// TIA Portal project "CMConstruccionesAutomatizacionHormigonera" (V16)

(* hardware
DEVICE "S7-1200 station_1"  S7-1200 Station
   slot 0: "Rack_0"  S7-1200 Rack  Rack  V1.0
   slot 1: "PLC_1"  CPU 1212C AC/DC/Rly  6ES7 212-1BE40-0XB0  V4.4
   slot 2: "DQ 8xRelay_1"  SM 1222 DQ8 x relay  6ES7 222-1HF32-0XB0  V2.0
*)

// ===== PLC "PLC_1"  CPU 1212C AC/DC/Rly =====

VAR_GLOBAL   // PLC tag table "Tabla de variables estándar"
   "Automatico" AT %I0.0 : Bool;
   "Sin Fin 1" AT %Q8.4 : Bool;
   "Start Cemento" AT %M0.0 : Bool;
   "Silo 1" AT %M0.1 : Bool;
   "Compuerta 1" AT %Q8.5 : Bool;
   "Silo 2" AT %M0.2 : Bool;
   "Compuerta 2" AT %Q0.5 : Bool;
   "Cemento listo" AT %M0.3 : Bool;
   "Input_Encoder" AT %ID1000 : DInt;
   "Comp Cemento listo" AT %Q8.0 : Bool;
   "Condiciones Cemento" AT %M0.4 : Bool;
   "Start Descarga" AT %M0.5 : Bool;
   "Piedra Listo" AT %M0.6 : Bool;
   "Compuerta 3" AT %Q0.0 : Bool;
   "Tag_1" AT %M0.7 : Bool;
   "Condiciones Piedra" AT %M3.0 : Bool;
   "Condiciones Arena" AT %M2.1 : Bool;
   "Compuerta 4" AT %Q0.2 : Bool;
   "Arena listo" AT %M2.2 : Bool;
   "Direccion encoder" AT %I0.2 : Bool;
   "Paso Piedra" AT %M2.3 : Bool;
   "Paso Arena" AT %M1.4 : Bool;
   "Start Agua" AT %M2.5 : Bool;
   "Condiciones Agua" AT %M1.6 : Bool;
   "Agua listo" AT %M1.7 : Bool;
   "Compresor" AT %Q8.3 : Bool;
   "Banda" AT %Q8.1 : Bool;
   "Agua" AT %Q8.2 : Bool;
   "Compuerta 5" AT %Q0.3 : Bool;
   "Paso Agua" AT %M2.0 : Bool;
   "System_Byte" AT %MB1 : Byte;
   "FirstScan" AT %M1.0 : Bool;
   "DiagStatusUpdate" AT %M1.1 : Bool;
   "AlwaysTRUE" AT %M1.2 : Bool;
   "AlwaysFALSE" AT %M1.3 : Bool;
   "System_Byte(1)" AT %MB2 : Byte;
   "Pulsos" AT %MD4 : DInt;
   "STATUS" AT %MW8 : Word;
   "Contador Agua" AT %I0.3 : Bool;
   "Salida Contador Agua" AT %MW10 : Word;
   "Ingreso Contador Agua" AT %MW12 : Word;
   "Compuerta 6" AT %Q0.4 : Bool;
   "reiniciar cemento" AT %M3.1 : Bool;
   "Tag_2" AT %M3.2 : Bool;
   "reiniciar aridos" AT %M3.3 : Bool;
   "Tag_3" AT %M3.4 : Bool;
   "arena paso" AT %M3.5 : Bool;
   "TiempoArena" AT %M3.6 : Bool;
   "fin cemento" AT %M3.7 : Bool;
   "tiempo banda" AT %M14.0 : Bool;
   "reserva" AT %M14.1 : Bool;
   "Compresor listo" AT %M14.2 : Bool;
   "fin aridos" AT %M14.3 : Bool;
   "Agua completa" AT %M14.4 : Bool;
   "Piedra 2" AT %Q0.1 : Bool;
END_VAR

// folder: System blocks/Program resources

DATA_BLOCK "IEC_Timer_0_DB"   // DB1
{ S7_Optimized_Access := 'TRUE' }
AUTHOR : Simatic
FAMILY : IEC
NAME : IEC_TMR
VERSION : 1.0
// stored: InstanceOfName IEC_TIMER
"IEC_TIMER"
BEGIN
END_DATA_BLOCK

DATA_BLOCK "IEC_Timer_0_DB_1"   // DB2
{ S7_Optimized_Access := 'TRUE' }
AUTHOR : Simatic
FAMILY : IEC
NAME : IEC_TMR
VERSION : 1.0
// stored: InstanceOfName IEC_TIMER
"IEC_TIMER"
BEGIN
END_DATA_BLOCK

DATA_BLOCK "IEC_Timer_0_DB_2"   // DB3
{ S7_Optimized_Access := 'TRUE' }
AUTHOR : Simatic
FAMILY : IEC
NAME : IEC_TMR
VERSION : 1.0
// stored: InstanceOfName IEC_TIMER
"IEC_TIMER"
BEGIN
END_DATA_BLOCK

DATA_BLOCK "IEC_Timer_0_DB_3"   // DB4
{ S7_Optimized_Access := 'TRUE' }
AUTHOR : Simatic
FAMILY : IEC
NAME : IEC_TMR
VERSION : 1.0
// stored: InstanceOfName IEC_TIMER
"IEC_TIMER"
BEGIN
END_DATA_BLOCK

DATA_BLOCK "IEC_Counter_0_DB"   // DB5
{ S7_Optimized_Access := 'TRUE' }
AUTHOR : Simatic
FAMILY : IEC
NAME : CNTR
VERSION : 1.0
// stored: InstanceOfName IEC_COUNTER
"IEC_COUNTER"
BEGIN
END_DATA_BLOCK

DATA_BLOCK "IEC_Timer_0_DB_4"   // DB6
{ S7_Optimized_Access := 'TRUE' }
AUTHOR : Simatic
FAMILY : IEC
NAME : IEC_TMR
VERSION : 1.0
// stored: InstanceOfName IEC_TIMER
"IEC_TIMER"
BEGIN
END_DATA_BLOCK

DATA_BLOCK "IEC_Timer_0_DB_5"   // DB7
{ S7_Optimized_Access := 'TRUE' }
AUTHOR : Simatic
FAMILY : IEC
NAME : IEC_TMR
VERSION : 1.0
// stored: InstanceOfName IEC_TIMER
"IEC_TIMER"
BEGIN
END_DATA_BLOCK

DATA_BLOCK "IEC_Timer_0_DB_6"   // DB8
{ S7_Optimized_Access := 'TRUE' }
AUTHOR : Simatic
FAMILY : IEC
NAME : IEC_TMR
VERSION : 1.0
// stored: InstanceOfName IEC_TIMER
"IEC_TIMER"
BEGIN
END_DATA_BLOCK

DATA_BLOCK "IEC_Timer_0_DB_7"   // DB9
{ S7_Optimized_Access := 'TRUE' }
AUTHOR : Simatic
FAMILY : IEC
NAME : IEC_TMR
VERSION : 1.0
// stored: InstanceOfName IEC_TIMER
"IEC_TIMER"
BEGIN
END_DATA_BLOCK

DATA_BLOCK "IEC_Timer_0_DB_8"   // DB10
{ S7_Optimized_Access := 'TRUE' }
AUTHOR : Simatic
FAMILY : IEC
NAME : IEC_TMR
VERSION : 1.0
// stored: InstanceOfName IEC_TIMER
"IEC_TIMER"
BEGIN
END_DATA_BLOCK

// folder: (top level)

ORGANIZATION_BLOCK "Main"   // OB1, LAD, ProgramCycle
TITLE = "Main Program Sweep (Cycle)"
{ S7_Optimized_Access := 'TRUE' }
VERSION : 0.1
   VAR_INPUT
      Initial_Call : Bool;   // Initial call of this OB
      Remanence : Bool;   // =True, if remanent data are available
   END_VAR
   VAR_TEMP   // added for the SCL form of the ladder/FBD networks
      _w1 : Bool;
      _w2 : Bool;
   END_VAR
BEGIN

REGION Network 1
   // Proceso Cemento
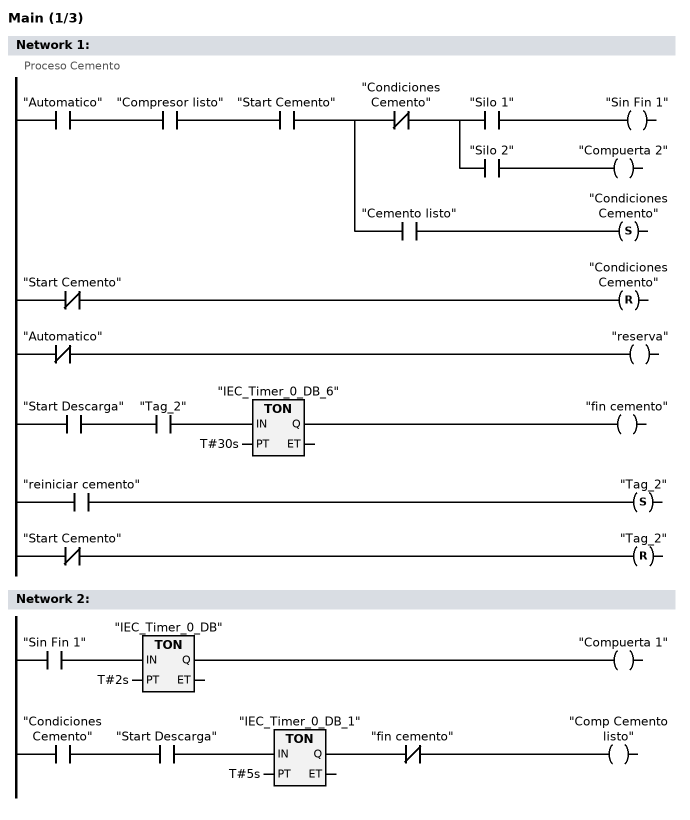
   #_w1 := "Automatico" AND "Compresor listo" AND "Start Cemento";
   #_w2 := #_w1 AND NOT "Condiciones Cemento";
   "Sin Fin 1" := #_w2 AND "Silo 1";
   "Compuerta 2" := #_w2 AND "Silo 2";
   IF #_w1 AND "Cemento listo" THEN "Condiciones Cemento" := TRUE; END_IF;
   IF NOT "Start Cemento" THEN "Condiciones Cemento" := FALSE; END_IF;
   "reserva" := NOT "Automatico";
   "IEC_Timer_0_DB_6".TON(IN := "Start Descarga" AND "Tag_2", PT := T#30s);
   "fin cemento" := "IEC_Timer_0_DB_6".Q;
   IF "reiniciar cemento" THEN "Tag_2" := TRUE; END_IF;
   IF NOT "Start Cemento" THEN "Tag_2" := FALSE; END_IF;
END_REGION

REGION Network 2
   "IEC_Timer_0_DB".TON(IN := "Sin Fin 1", PT := T#2s);
   "Compuerta 1" := "IEC_Timer_0_DB".Q;
   "IEC_Timer_0_DB_1".TON(IN := "Condiciones Cemento" AND "Start Descarga", PT := T#5s);
   "Comp Cemento listo" := "IEC_Timer_0_DB_1".Q AND NOT "fin cemento";
END_REGION

REGION Network 3
   // Proceso Aridos
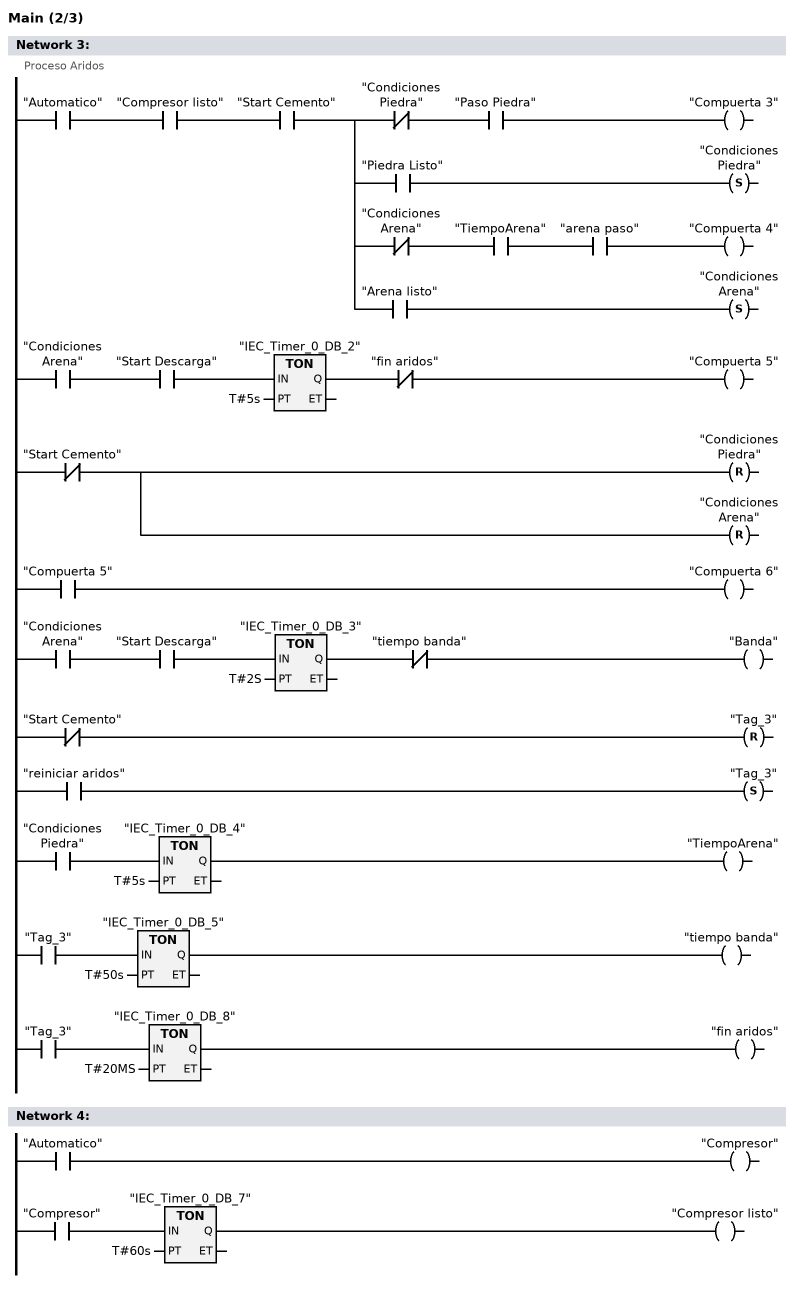
   #_w1 := "Automatico" AND "Compresor listo" AND "Start Cemento";
   "Compuerta 3" := #_w1 AND NOT "Condiciones Piedra" AND "Paso Piedra";
   IF #_w1 AND "Piedra Listo" THEN "Condiciones Piedra" := TRUE; END_IF;
   "Compuerta 4" := #_w1 AND NOT "Condiciones Arena" AND "TiempoArena" AND "arena paso";
   IF #_w1 AND "Arena listo" THEN "Condiciones Arena" := TRUE; END_IF;
   "IEC_Timer_0_DB_2".TON(IN := "Condiciones Arena" AND "Start Descarga", PT := T#5s);
   "Compuerta 5" := "IEC_Timer_0_DB_2".Q AND NOT "fin aridos";
   IF NOT "Start Cemento" THEN
       "Condiciones Piedra" := FALSE;
       "Condiciones Arena" := FALSE;
   END_IF;
   "Compuerta 6" := "Compuerta 5";
   "IEC_Timer_0_DB_3".TON(IN := "Condiciones Arena" AND "Start Descarga", PT := T#2S);
   "Banda" := "IEC_Timer_0_DB_3".Q AND NOT "tiempo banda";
   IF NOT "Start Cemento" THEN "Tag_3" := FALSE; END_IF;
   IF "reiniciar aridos" THEN "Tag_3" := TRUE; END_IF;
   "IEC_Timer_0_DB_4".TON(IN := "Condiciones Piedra", PT := T#5s);
   "TiempoArena" := "IEC_Timer_0_DB_4".Q;
   "IEC_Timer_0_DB_5".TON(IN := "Tag_3", PT := T#50s);
   "tiempo banda" := "IEC_Timer_0_DB_5".Q;
   "IEC_Timer_0_DB_8".TON(IN := "Tag_3", PT := T#20MS);
   "fin aridos" := "IEC_Timer_0_DB_8".Q;
END_REGION

REGION Network 4
   "Compresor" := "Automatico";
   "IEC_Timer_0_DB_7".TON(IN := "Compresor", PT := T#60s);
   "Compresor listo" := "IEC_Timer_0_DB_7".Q;
END_REGION

REGION Network 5
   // Proceso Agua
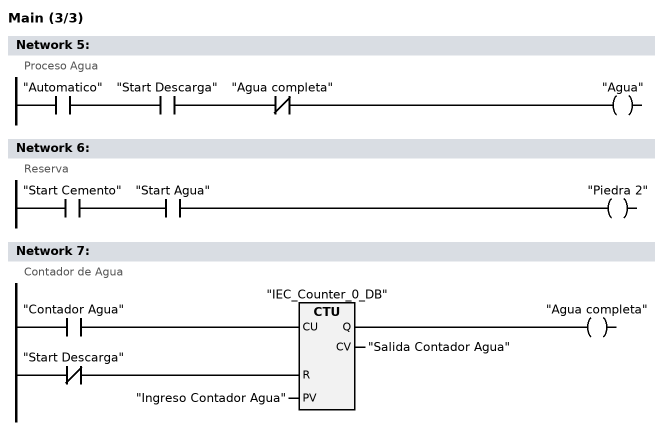
   RUNG wire#powerrail
      Contact( "Automatico" )
      Contact( "Start Descarga" )
      I_Contact( "Agua completa" )
      Coil( "Agua" )
   END_RUNG
   // the same network as SCL:
   "Agua" := "Automatico" AND "Start Descarga" AND NOT "Agua completa";
END_REGION

REGION Network 6
   // Reserva
   RUNG wire#powerrail
      Contact( "Start Cemento" )
      Contact( "Start Agua" )
      Coil( "Piedra 2" )
   END_RUNG
   // the same network as SCL:
   "Piedra 2" := "Start Cemento" AND "Start Agua";
END_REGION

REGION Network 7
   // Contador de Agua
   "IEC_Counter_0_DB".CTU(CU := "Contador Agua",
                          R := NOT "Start Descarga",
                          PV := "Ingreso Contador Agua",
                          CV => "Salida Contador Agua");
   "Agua completa" := "IEC_Counter_0_DB".Q;
END_REGION
END_ORGANIZATION_BLOCK